(* Logix 5000 project; controller pracainz_ne 1769-L16ER-BB1B rev 30.11; software revision 30.00 *)

TASK MainTask (continuous, watchdog 500 ms) : MainProgram

MODULES
   Local : 1769-L16ER-BB1B (PointIO 0, rev 30.11)
      PF525_1 : vendor 1 type 151 code 9 (Ethernet 192.168.1.76, rev 4.1, Output RPI 20 ms)
          : vendor 1 type 151 code 1566 (DSI 2, rev 1.1)
      pointio : 1734-AENTR (Ethernet 192.168.1.74, rev 5.1, Output RPI 20 ms)
         RTD : 1734-IR2 (PointIO 5, rev 3.1, Input RPI 80 ms)
         input_2 : 1734-IB8 (PointIO 4, rev 3.1)
         input_1 : 1734-IB8 (PointIO 3, rev 3.1)
         potenc : 1734-IE2V (PointIO 6, rev 3.1, Input RPI 80 ms)
         output_2 : 1734-OB8 (PointIO 2, rev 3.1)
         output_1 : 1734-OB8 (PointIO 1, rev 3.1)
      Discrete_IO : Embedded (PointIO 1, rev 30.11, Output RPI 200 ms)
END_MODULES

VAR_GLOBAL   (* controller tags *)
   AUTO_1 : BOOL;
   auto_once : BOOL;
   BELT_CONV_2_0_1_L : BOOL;
   BELT_CONV_2_0_1_U : BOOL;
   BELT_CONV_2_0_2_L : BOOL;
   BELT_CONV_2_0_2_U : BOOL;
   BELT_CONV_2_1_1 : BOOL;
   BELT_CONV_2_1_1_L : BOOL;
   BELT_CONV_2_1_1_U : BOOL;
   BELT_CONV_2_1_2 : BOOL;
   BELT_CONV_2_1_2_L : BOOL;
   BELT_CONV_2_1_2_U : BOOL;
   BELT_CONV_4_0_1_L : BOOL;
   BELT_CONV_4_0_1_U : BOOL;
   BELT_CONV_4_0_2_L : BOOL;
   BELT_CONV_4_0_2_U : BOOL;
   BELT_CONV_4_1_1_L : BOOL;
   BELT_CONV_4_1_1_U : BOOL;
   BELT_CONV_4_1_2_L : BOOL;
   BELT_CONV_4_1_2_U : BOOL;
   BOOL_IN_0 : BOOL;
   BOOL_IN_1 : BOOL;
   BOOL_IN_10 : BOOL;
   BOOL_IN_11 : BOOL := 1;
   BOOL_IN_12 : BOOL := 1;
   BOOL_IN_13 : BOOL := 1;
   BOOL_IN_14 : BOOL := 1;
   BOOL_IN_15 : BOOL := 1;
   BOOL_IN_16 : BOOL;
   BOOL_IN_17 : BOOL;
   BOOL_IN_18 : BOOL := 1;
   BOOL_IN_19 : BOOL := 1;
   BOOL_IN_2 : BOOL;
   BOOL_IN_20 : BOOL;
   BOOL_IN_21 : BOOL;
   BOOL_IN_22 : BOOL := 1;
   BOOL_IN_23 : BOOL;
   BOOL_IN_24 : BOOL;
   BOOL_IN_25 : BOOL;
   BOOL_IN_26 : BOOL := 1;
   BOOL_IN_27 : BOOL := 1;
   BOOL_IN_28 : BOOL;
   BOOL_IN_29 : BOOL := 1;
   BOOL_IN_3 : BOOL;
   BOOL_IN_30 : BOOL := 1;
   BOOL_IN_31 : BOOL := 1;
   BOOL_IN_32 : BOOL := 1;
   BOOL_IN_33 : BOOL := 1;
   BOOL_IN_34 : BOOL;
   BOOL_IN_35 : BOOL;
   BOOL_IN_36 : BOOL;
   BOOL_IN_37 : BOOL;
   BOOL_IN_38 : BOOL := 1;
   BOOL_IN_39 : BOOL := 1;
   BOOL_IN_4 : BOOL;
   BOOL_IN_40 : BOOL := 1;
   BOOL_IN_41 : BOOL;
   BOOL_IN_42 : BOOL;
   BOOL_IN_43 : BOOL;
   BOOL_IN_5 : BOOL;
   BOOL_IN_6 : BOOL;
   BOOL_IN_7 : BOOL;
   BOOL_IN_8 : BOOL := 1;
   BOOL_IN_9 : BOOL;
   BOOL_OUT_0 : BOOL;
   BOOL_OUT_1 : BOOL;
   BOOL_OUT_10 : BOOL;
   BOOL_OUT_11 : BOOL;
   BOOL_OUT_12 : BOOL;
   BOOL_OUT_13 : BOOL;
   BOOL_OUT_14 : BOOL;
   BOOL_OUT_15 : BOOL;
   BOOL_OUT_16 : BOOL;
   BOOL_OUT_17 : BOOL;
   BOOL_OUT_18 : BOOL;
   BOOL_OUT_19 : BOOL;
   BOOL_OUT_2 : BOOL;
   BOOL_OUT_20 : BOOL;
   BOOL_OUT_21 : BOOL;
   BOOL_OUT_22 : BOOL;
   BOOL_OUT_23 : BOOL;
   BOOL_OUT_24 : BOOL;
   BOOL_OUT_25 : BOOL;
   BOOL_OUT_26 : BOOL;
   BOOL_OUT_27 : BOOL;
   BOOL_OUT_28 : BOOL;
   BOOL_OUT_29 : BOOL;
   BOOL_OUT_3 : BOOL;
   BOOL_OUT_30 : BOOL;
   BOOL_OUT_31 : BOOL;
   BOOL_OUT_32 : BOOL;
   BOOL_OUT_33 : BOOL;
   BOOL_OUT_34 : BOOL;
   BOOL_OUT_35 : BOOL := 1;
   BOOL_OUT_36 : BOOL := 1;
   BOOL_OUT_37 : BOOL;
   BOOL_OUT_38 : BOOL;
   BOOL_OUT_39 : BOOL;
   BOOL_OUT_4 : BOOL;
   BOOL_OUT_40 : BOOL;
   BOOL_OUT_41 : BOOL;
   BOOL_OUT_42 : BOOL;
   BOOL_OUT_43 : BOOL;
   BOOL_OUT_44 : BOOL;
   BOOL_OUT_45 : BOOL;
   BOOL_OUT_46 : BOOL;
   BOOL_OUT_47 : BOOL;
   BOOL_OUT_48 : BOOL;
   BOOL_OUT_49 : BOOL := 1;
   BOOL_OUT_5 : BOOL;
   BOOL_OUT_50 : BOOL;
   BOOL_OUT_51 : BOOL;
   BOOL_OUT_52 : BOOL;
   BOOL_OUT_53 : BOOL;
   BOOL_OUT_54 : BOOL;
   BOOL_OUT_55 : BOOL;
   BOOL_OUT_56 : BOOL;
   BOOL_OUT_57 : BOOL;
   BOOL_OUT_58 : BOOL;
   BOOL_OUT_6 : BOOL;
   BOOL_OUT_7 : BOOL;
   BOOL_OUT_8 : BOOL;
   BOOL_OUT_9 : BOOL;
   CHAIN_1 : BOOL;
   CHAIN_1_B : BOOL;
   CHAIN_1_F : BOOL;
   CHAIN_1_L : BOOL;
   CHAIN_1_R : BOOL;
   CHAIN_2 : BOOL;
   CHAIN_2_B : BOOL;
   CHAIN_2_F : BOOL;
   CHAIN_2_L : BOOL;
   CHAIN_2_R : BOOL;
   CLAMPED : BOOL;
   CLAMPED_R : BOOL;
   COUNT_R : DINT;
   dokonczyc : BOOL;
   EMERGENCY_ALL : BOOL := 1;
   END : BOOL;
   END_OF_DAY : BOOL;
   FLOAT_IN_0 : REAL := 1.0;
   FLOAT_IN_1 : REAL := 3.50007;
   FLOAT_IN_2 : REAL := 6.000015;
   FLOAT_IN_3 : REAL := 5.000424;
   FLOAT_IN_4 : REAL := 3.999957;
   FLOAT_IN_5 : REAL := 4.999908;
   FLOAT_IN_6 : REAL;
   FLOAT_OUT_0 : REAL := 6.000015;
   FLOAT_OUT_1 : REAL := 4.999908;
   FLOAT_OUT_2 : REAL := 3.50007;
   FLOAT_OUT_3 : REAL := 3.999957;
   FLOAT_OUT_4 : REAL := 5.000424;
   FLOAT_OUT_5 : REAL;
   FLOAT_OUT_6 : REAL;
   FLOAT_OUT_7 : REAL;
   full_palet : BOOL;
   FULL_PALET_R : BOOL;
   GGG : BOOL;
   height : BOOL;
   height1 : BOOL;
   HHH : BOOL;
   Input_1 : BOOL;
   Input_1_R : BOOL;
   Input_2 : BOOL;
   Input_2_R : BOOL;
   Input_3 : BOOL;
   Input_3_R : BOOL;
   Input_4 : BOOL;
   Input_4_R : BOOL;
   Input_5 : BOOL;
   Input_5_R : BOOL;
   Input_6 : BOOL;
   Input_6_R : BOOL;
   Input_7 : BOOL;
   Input_7_R : BOOL;
   INT_IN_0 : INT;
   INT_IN_1 : INT := 99;
   INT_IN_2 : INT;
   INT_IN_3 : INT;
   INT_OUT_0 : INT;
   koniec : BOOL;
   LATCH_MANUAL : BOOL;
   LEFT_PACK : BOOL;
   LEFT_PACKED : BOOL;
   LEFT_PICK : BOOL;
   LEWA_LINIA : BOOL;
   LEWA_STRONA : BOOL;
   M_01 : BOOL := 1;
   M_02 : BOOL := 1;
   M_03 : BOOL;
   M_04 : BOOL;
   M_05 : BOOL;
   M_06 : BOOL;
   M_07 : BOOL;
   M_08 : BOOL;
   M_09 : BOOL;
   M_10 : BOOL;
   M_11 : BOOL;
   M_12 : BOOL;
   M_13 : BOOL;
   M_14 : BOOL;
   M_15 : BOOL;
   M_16 : BOOL;
   M_17 : BOOL;
   M_18 : BOOL;
   M_19 : BOOL;
   M_20 : BOOL;
   M_21 : INT;
   M_22 : INT;
   M_23 : BOOL;
   M_24 : BOOL;
   M_25 : BOOL := 1;
   M_26 : BOOL;
   M_27 : BOOL;
   M_28 : BOOL;
   M_29 : BOOL;
   M_30 : BOOL;
   M_31 : BOOL;
   M_32 : BOOL;
   M_33 : BOOL;
   M_34 : BOOL;
   M_35 : BOOL;
   M_36 : BOOL;
   M_37 : BOOL;
   M_38 : BOOL;
   M_39 : BOOL;
   M_40 : BOOL;
   M_41 : BOOL;
   M_42 : BOOL;
   M_43 : BOOL;
   M_44 : BOOL;
   M_45 : BOOL;
   M_46 : BOOL;
   M_47 : BOOL;
   MANUAL_ALL : BOOL;
   manual_once : BOOL;
   OSF_03_O : BOOL;
   OSF_03_S : BOOL;
   OSF_05 : BOOL;
   OSF_10_O : BOOL;
   OSF_10_S : BOOL;
   OSF_11_O : BOOL;
   OSF_11_S : BOOL;
   OSFI_01 : DINT;
   OSR_10_O : BOOL;
   OSR_10_S : BOOL := 1;
   OSR_13_O : BOOL;
   OSR_13_S : BOOL;
   OSR_14_O : BOOL;
   OSR_14_S : BOOL := 1;
   OSR_15_O : BOOL;
   OSR_15_S : BOOL;
   OSR_16_O : BOOL;
   OSR_16_S : BOOL;
   OSR_17_O : BOOL;
   OSR_17_S : BOOL;
   OSR_18_O : BOOL;
   OSR_18_S : BOOL := 1;
   OSR_19_O : BOOL;
   OSR_19_S : BOOL;
   OSR_20_O : BOOL;
   OSR_20_S : BOOL;
   OSR_21_O : BOOL;
   OSR_21_S : BOOL := 1;
   OSR_Auto_O : BOOL;
   OSR_Auto_S : BOOL;
   P_P_0_X_D : REAL;
   P_P_0_Y_D : REAL;
   P_P_0_Z_D : REAL;
   PICK : BOOL := 1;
   PRAWA_LINIA : BOOL;
   PRAWA_STRONA : BOOL;
   PUSHER_2 : BOOL;
   READY_L : BOOL;
   READY_R : BOOL;
   Reset : BOOL;
   RESET_1 : BOOL;
   reset_timer : BOOL;
   reset_timer_l : BOOL;
   RIGHT_PACK : BOOL;
   RIGHT_PICK : BOOL;
   ROLL_1 : BOOL;
   ROLL_2 : BOOL;
   ROLL_3 : BOOL;
   ROLL_4 : BOOL;
   ROLL_5 : BOOL;
   ROLL_6 : BOOL;
   ROLL_7 : BOOL;
   START : BOOL;
   START_ALL : BOOL;
   STOP_LEFT : BOOL;
   STOP_RIGHT : BOOL;
   stop_work_timer : TIMER := (PRE := 60000, ACC := 3399, EN := 1, TT := 1);
   stop_work_timer_2 : TIMER := (PRE := 60000);
   stopped_left : BOOL;
   stopped_right : BOOL;
   TASMA_1_P : BOOL;
   TASMA_2_P : BOOL;
   TASMA_5_P : BOOL;
   TASMA_9_P : BOOL;
   TEST_HH : BOOL := 1;
   TIMER_1 : TIMER := (PRE := 800);
   TIMER_2 : TIMER := (PRE := 10000, ACC := 10000, DN := 1);
   TIMER_3_R : TIMER := (PRE := 10000, ACC := 10000, DN := 1);
   TIMER_left : TIMER := (PRE := 100);
   TIMER_LEFT_P_P : TIMER := (PRE := 4000);
   TIMER_PALET : TIMER := (PRE := 500);
   timer_right : TIMER := (PRE := 2000);
   TIMER_RIGHT_P_P : TIMER := (PRE := 4000);
   timer_state_1 : BOOL;
   timer_state_2 : BOOL;
   timer_state_3 : BOOL;
   timer_state_4 : BOOL;
   timer_state_5 : BOOL;
   ton1 : TIMER := (PRE := 2000, ACC := 2000, DN := 1);
   TON1_R : TIMER := (PRE := 2000, ACC := 2000, DN := 1);
   ton2 : TIMER := (PRE := 2000, ACC := 2000, DN := 1);
   TON2_R : TIMER := (PRE := 2000, ACC := 2000, DN := 1);
   ton3 : TIMER := (PRE := 2000);
   ton3_R : TIMER := (PRE := 2000);
   ton4 : TIMER := (PRE := 1000);
   TON4_R : TIMER := (PRE := 1000);
   ton5 : TIMER := (PRE := 3000);
   TON5_R : TIMER := (PRE := 3000);
   ton6 : TIMER := (PRE := 1000);
   TON6_R : TIMER := (PRE := 2000);
   TON7 : TIMER := (PRE := 2000);
   TON7_R : TIMER := (PRE := 2000);
   TONR_01 : FBD_TIMER;
   TONR_02 : FBD_TIMER;
   TONR_03 : FBD_TIMER;
   TONR_04 : FBD_TIMER;
   TONR_05 : FBD_TIMER;
   wait_left : BOOL;
   X0 : REAL := 3.5;
   X1 : REAL := 5.29;
   Y0 : REAL := 6.0;
   Y1 : REAL := 3.8;
   ZNIENNA : BOOL;
END_VAR

PROGRAM MainProgram   (* main routine MainRoutine *)
VAR
   AUTO : ALIAS FOR M_03;
   BELT_CONV_2_0 : ALIAS FOR BOOL_OUT_0;
   BELT_CONV_2_1 : ALIAS FOR BOOL_OUT_1;
   BELT_CONV_2_2 : ALIAS FOR BOOL_OUT_2;
   BELT_CONV_2_3 : ALIAS FOR BOOL_OUT_3;
   BELT_CONV_2_4 : ALIAS FOR BOOL_OUT_4;
   BELT_CONV_2_5 : ALIAS FOR BOOL_OUT_5;
   BELT_CONV_2_6 : ALIAS FOR BOOL_OUT_6;
   BELT_CONV_2_7 : ALIAS FOR BOOL_OUT_7;
   BELT_CONV_2_CCW : ALIAS FOR BOOL_OUT_27;
   BELT_CONV_4_0 : ALIAS FOR BOOL_OUT_8;
   BELT_CONV_4_1 : ALIAS FOR BOOL_OUT_9;
   BELT_CONV_4_2 : ALIAS FOR BOOL_OUT_10;
   BELT_CONV_4_3 : ALIAS FOR BOOL_OUT_11;
   BELT_CONV_CCW_0 : ALIAS FOR BOOL_OUT_23;
   BELT_CONV_CCW_3 : ALIAS FOR BOOL_OUT_24;
   BELT_CONV_CCW_4 : ALIAS FOR BOOL_OUT_25;
   BELT_CONV_CW_0 : ALIAS FOR BOOL_OUT_26;
   BELT_CONV_CW_1 : ALIAS FOR BOOL_OUT_20;
   BELT_CONV_CW_2 : ALIAS FOR BOOL_OUT_21;
   BELT_CONV_CW_5 : ALIAS FOR BOOL_OUT_22;
   BTN_RESET : ALIAS FOR BOOL_IN_34;
   BTN_START : ALIAS FOR BOOL_IN_35;
   BTN_STOP : ALIAS FOR BOOL_IN_38;
   CAP_SEN_0 : ALIAS FOR BOOL_IN_0;
   CAP_SEN_1 : ALIAS FOR BOOL_IN_1;
   CAP_SEN_2 : ALIAS FOR BOOL_IN_2;
   CAP_SEN_3 : ALIAS FOR BOOL_IN_3;
   CHAIN_0_LEFT : ALIAS FOR BOOL_OUT_16;
   CHAIN_0_N : ALIAS FOR BOOL_OUT_13;
   CHAIN_0_P : ALIAS FOR BOOL_OUT_12;
   CHAIN_0_RIGHT : ALIAS FOR BOOL_OUT_18;
   CHAIN_1_LEFT : ALIAS FOR BOOL_OUT_17;
   CHAIN_1_N : ALIAS FOR BOOL_OUT_15;
   CHAIN_1_P : ALIAS FOR BOOL_OUT_14;
   CHAIN_1_RIGHT : ALIAS FOR BOOL_OUT_19;
   CNC_0_START : ALIAS FOR BOOL_OUT_38;
   CNC_1_START : ALIAS FOR BOOL_OUT_40;
   CNC_RESET : BOOL;
   CNC_START_1 : BOOL;
   CNC_STOP_1 : BOOL;
   COUNT : DINT;
   DIFF_SEN_0 : ALIAS FOR BOOL_IN_4;
   DIFF_SEN_1 : ALIAS FOR BOOL_IN_5;
   DIFF_SEN_2 : ALIAS FOR BOOL_IN_6;
   DIFF_SEN_3 : ALIAS FOR BOOL_IN_7;
   DIFF_SEN_4 : ALIAS FOR BOOL_IN_8;
   EMERGENCY : ALIAS FOR BOOL_IN_33;
   emergency_disp : BOOL;
   EMIT_0 : ALIAS FOR BOOL_OUT_28;
   EMIT_1 : ALIAS FOR BOOL_OUT_29;
   EMIT_2 : ALIAS FOR BOOL_OUT_30;
   EMIT_3 : ALIAS FOR BOOL_OUT_31;
   FREQUENCY : INT := 3000;
   GREEN_B : ALIAS FOR M_22;
   GREEN_L : ALIAS FOR M_21;
   koniecpracy : ALIAS FOR koniec;
   MACH_CEN_0_LIDS : ALIAS FOR BOOL_OUT_41;
   MACH_CEN_0_PROGRESS : ALIAS FOR INT_IN_0;
   MACH_CEN_0_RESET : ALIAS FOR BOOL_OUT_39;
   MACH_CEN_0_START : ALIAS FOR BOOL_OUT_37;
   MACH_CEN_0_STOP : ALIAS FOR BOOL_OUT_35;
   MACH_CEN_1_LIDS : ALIAS FOR BOOL_OUT_42;
   MACH_CEN_1_PROGRESS : ALIAS FOR INT_IN_1;
   MACH_CEN_1_RESET : ALIAS FOR BOOL_OUT_40;
   MACH_CEN_1_START : ALIAS FOR BOOL_OUT_38;
   MACH_CEN_1_STOP : ALIAS FOR BOOL_OUT_36;
   MACHI_CE_0_BUSY : ALIAS FOR BOOL_IN_14;
   MACHI_CE_0_ERR : ALIAS FOR BOOL_IN_16;
   MACHI_CE_0_OPEN : ALIAS FOR BOOL_IN_12;
   MACHI_CE_1_BUSY : ALIAS FOR BOOL_IN_15;
   MACHI_CE_1_ERR : ALIAS FOR BOOL_IN_17;
   MACHI_CE_1_OPEN : ALIAS FOR BOOL_IN_13;
   MACHINE_X : REAL;
   MACHINE_Y : REAL;
   MACHINE_Z : REAL;
   MANUAL : ALIAS FOR M_04;
   manual_disp : BOOL := 1;
   MOVE : ALIAS FOR M_16;
   NOT_BLUE : ALIAS FOR M_24;
   NOT_GREEN : ALIAS FOR M_23;
   OSF_01_O : ALIAS FOR M_07;
   OSF_01_S : ALIAS FOR M_06;
   OSF_02_O : ALIAS FOR M_11;
   OSF_02_S : ALIAS FOR M_10;
   OSF_03_O : ALIAS FOR M_05;
   OSF_03_S : ALIAS FOR M_25;
   OSF_04_O : ALIAS FOR M_26;
   OSF_04_S : ALIAS FOR M_27;
   OSF_05_O : ALIAS FOR M_28;
   OSF_05_S : ALIAS FOR M_29;
   OSF_06_O : ALIAS FOR M_30;
   OSF_06_S : ALIAS FOR M_31;
   OSF_07_O : ALIAS FOR M_32;
   OSF_07_S : ALIAS FOR M_30;
   OSF_08_O : ALIAS FOR M_41;
   OSF_08_S : ALIAS FOR M_42;
   OSF_09_O : BOOL;
   OSF_09_S : BOOL := 1;
   OSR_01_O : ALIAS FOR M_09;
   OSR_01_S : ALIAS FOR M_08;
   OSR_02_O : ALIAS FOR M_13;
   OSR_02_S : ALIAS FOR M_12;
   OSR_03_O : ALIAS FOR M_17;
   OSR_03_S : ALIAS FOR M_18;
   OSR_04_O : ALIAS FOR M_19;
   OSR_04_S : ALIAS FOR M_20;
   OSR_05_O : ALIAS FOR M_14;
   OSR_05_S : ALIAS FOR M_15;
   OSR_06_O : ALIAS FOR M_33;
   OSR_06_S : ALIAS FOR M_34;
   OSR_07_O : ALIAS FOR M_35;
   OSR_07_S : ALIAS FOR M_36;
   OSR_08_O : ALIAS FOR M_37;
   OSR_08_S : ALIAS FOR M_38;
   OSR_09_O : ALIAS FOR M_39;
   OSR_09_S : ALIAS FOR M_40;
   P_P_0_C_LIMIT : ALIAS FOR BOOL_IN_18;
   P_P_0_CP : ALIAS FOR BOOL_OUT_43;
   P_P_0_DETE : ALIAS FOR BOOL_IN_20;
   P_P_0_GRAB : ALIAS FOR BOOL_OUT_45;
   P_P_0_X : ALIAS FOR FLOAT_OUT_2;
   P_P_0_X_POSITION : ALIAS FOR FLOAT_IN_1;
   P_P_0_Y : ALIAS FOR FLOAT_OUT_0;
   P_P_0_Y_POSITION : ALIAS FOR FLOAT_IN_2;
   P_P_0_Z : ALIAS FOR FLOAT_OUT_4;
   P_P_0_Z_POSITION : ALIAS FOR FLOAT_IN_3;
   P_P_1_C_LIMIT : ALIAS FOR BOOL_IN_19;
   P_P_1_CP : ALIAS FOR BOOL_OUT_44;
   P_P_1_DETE : ALIAS FOR BOOL_IN_21;
   P_P_1_GRAB : ALIAS FOR BOOL_OUT_46;
   P_P_1_X : ALIAS FOR FLOAT_OUT_3;
   P_P_1_X_D : REAL := 4.0;
   P_P_1_X_POSITION : ALIAS FOR FLOAT_IN_4;
   P_P_1_Y : ALIAS FOR FLOAT_OUT_1;
   P_P_1_Y_D : REAL := 5.0;
   P_P_1_Y_POSITION : ALIAS FOR FLOAT_IN_5;
   P_P_1_Z : ALIAS FOR FLOAT_OUT_5;
   P_P_1_Z_D : REAL := 5.0;
   P_P_1_Z_POSITION : ALIAS FOR FLOAT_IN_6;
   PUSH_0 : ALIAS FOR BOOL_OUT_47;
   PUSH_0_BACK : ALIAS FOR BOOL_IN_22;
   PUSH_0_FRONT : ALIAS FOR BOOL_IN_23;
   PUSH_1 : ALIAS FOR BOOL_OUT_48;
   PUSH_1_BACK : ALIAS FOR BOOL_IN_39;
   PUSH_1_FRONT : ALIAS FOR BOOL_IN_24;
   PUSHER_1 : BOOL;
   REMOVER : ALIAS FOR BOOL_OUT_49;
   RETRO_SEN_0 : ALIAS FOR BOOL_IN_25;
   RETRO_SEN_1 : ALIAS FOR BOOL_IN_26;
   RETRO_SEN_2 : ALIAS FOR BOOL_IN_27;
   RETRO_SEN_3 : ALIAS FOR BOOL_IN_28;
   RETRO_SEN_4 : ALIAS FOR BOOL_IN_29;
   RETRO_SEN_5 : ALIAS FOR BOOL_IN_30;
   RETRO_SEN_6 : ALIAS FOR BOOL_IN_31;
   RETRO_SEN_7 : ALIAS FOR BOOL_IN_32;
   ROLL_4_0 : ALIAS FOR BOOL_OUT_50;
   ROLL_4_1 : ALIAS FOR BOOL_OUT_51;
   ROLL_4_2 : ALIAS FOR BOOL_OUT_52;
   ROLL_6_0 : ALIAS FOR BOOL_OUT_53;
   ROLL_6_1 : ALIAS FOR BOOL_OUT_54;
   start_disp : BOOL := 1;
   STOP_ALL : ALIAS FOR M_02;
   stop_disp : BOOL;
   STOP_EMIT : ALIAS FOR M_01;
   TASMA_1 : BOOL;
   TASMA_10 : BOOL;
   TASMA_2 : BOOL;
   TASMA_3 : BOOL;
   TASMA_4 : BOOL;
   TASMA_5 : BOOL;
   TASMA_6 : BOOL;
   TASMA_7 : BOOL;
   TASMA_8 : BOOL;
   TASMA_9 : BOOL;
   VISION_SEN_0 : ALIAS FOR INT_IN_2;
   VISION_SEN_1 : ALIAS FOR INT_IN_3;
END_VAR

ROUTINE MainRoutine   (* ladder *)
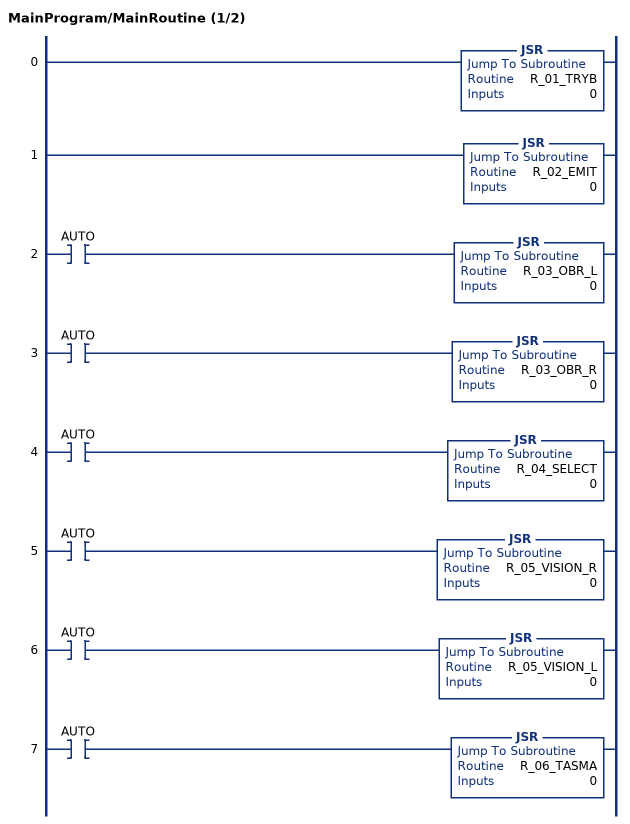
   0: JSR(R_01_TRYB,0);
   1: JSR(R_02_EMIT,0);
   2: XIC(AUTO)JSR(R_03_OBR_L,0);
   3: XIC(AUTO)JSR(R_03_OBR_R,0);
   4: XIC(AUTO)JSR(R_04_SELECT,0);
   5: XIC(AUTO)JSR(R_05_VISION_R,0);
   6: XIC(AUTO)JSR(R_05_VISION_L,0);
   7: XIC(AUTO)JSR(R_06_TASMA,0);
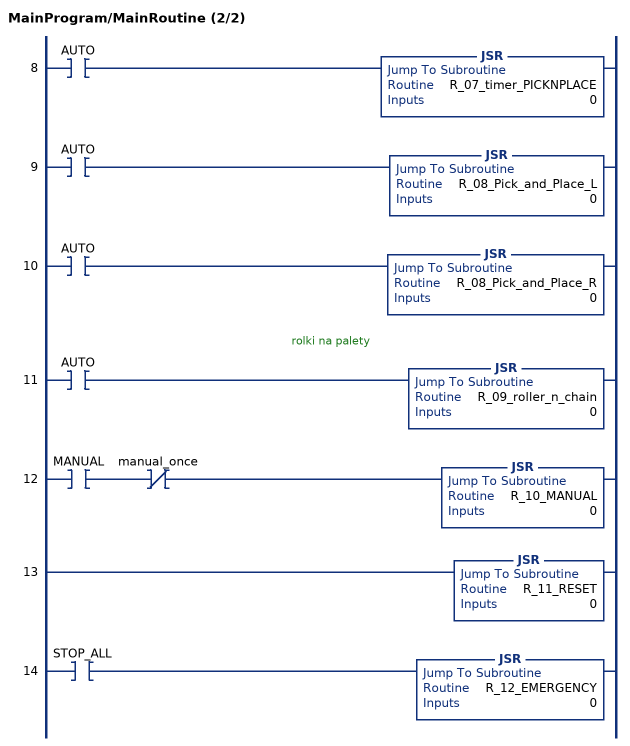
   8: XIC(AUTO)JSR(R_07_timer_PICKNPLACE,0);
   9: XIC(AUTO)JSR(R_08_Pick_and_Place_L,0);
   10: XIC(AUTO)JSR(R_08_Pick_and_Place_R,0);
   // rolki na palety
   11: XIC(AUTO)JSR(R_09_roller_n_chain,0);
   12: XIC(MANUAL)XIO(manual_once)JSR(R_10_MANUAL,0);
   13: JSR(R_11_RESET,0);
   14: XIC(STOP_ALL)JSR(R_12_EMERGENCY,0);
END_ROUTINE

ROUTINE R_01_TRYB   (* ladder *)
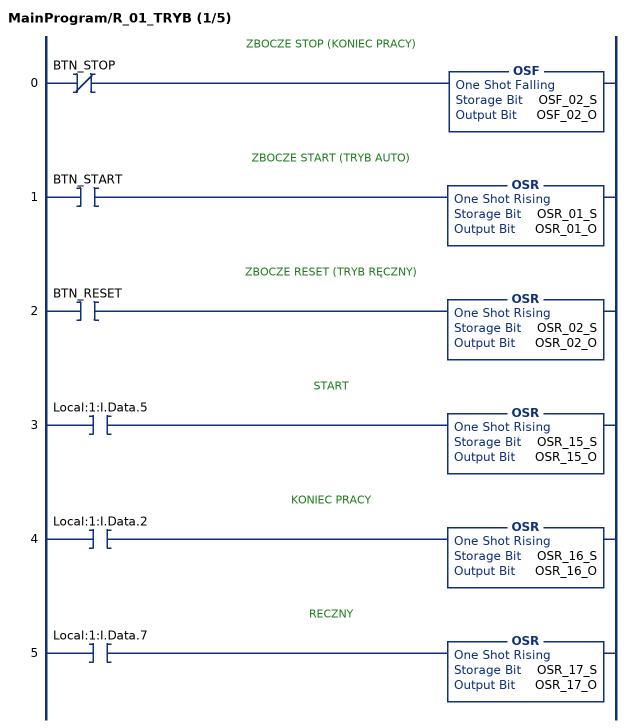
   // ZBOCZE STOP (KONIEC PRACY)
   0: XIO(BTN_STOP)OSF(OSF_02_S,OSF_02_O);
   // ZBOCZE START (TRYB AUTO)
   1: XIC(BTN_START)OSR(OSR_01_S,OSR_01_O);
   // ZBOCZE RESET (TRYB RĘCZNY)
   2: XIC(BTN_RESET)OSR(OSR_02_S,OSR_02_O);
   // START
   3: XIC(Local:1:I.Data.5)OSR(OSR_15_S,OSR_15_O);
   // KONIEC PRACY
   4: XIC(Local:1:I.Data.2)OSR(OSR_16_S,OSR_16_O);
   // RECZNY
   5: XIC(Local:1:I.Data.7)OSR(OSR_17_S,OSR_17_O);
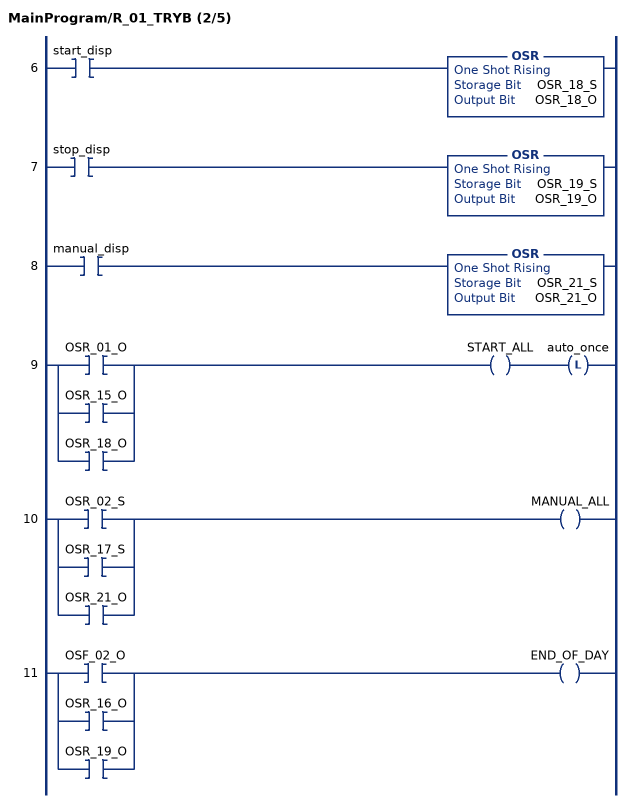
   6: XIC(start_disp)OSR(OSR_18_S,OSR_18_O);
   7: XIC(stop_disp)OSR(OSR_19_S,OSR_19_O);
   8: XIC(manual_disp)OSR(OSR_21_S,OSR_21_O);
   9: [XIC(OSR_01_O) ,XIC(OSR_15_O) ,XIC(OSR_18_O) ]OTE(START_ALL)OTL(auto_once);
   10: [XIC(OSR_02_S) ,XIC(OSR_17_S) ,XIC(OSR_21_O) ]OTE(MANUAL_ALL);
   11: [XIC(OSF_02_O) ,XIC(OSR_16_O) ,XIC(OSR_19_O) ]OTE(END_OF_DAY);
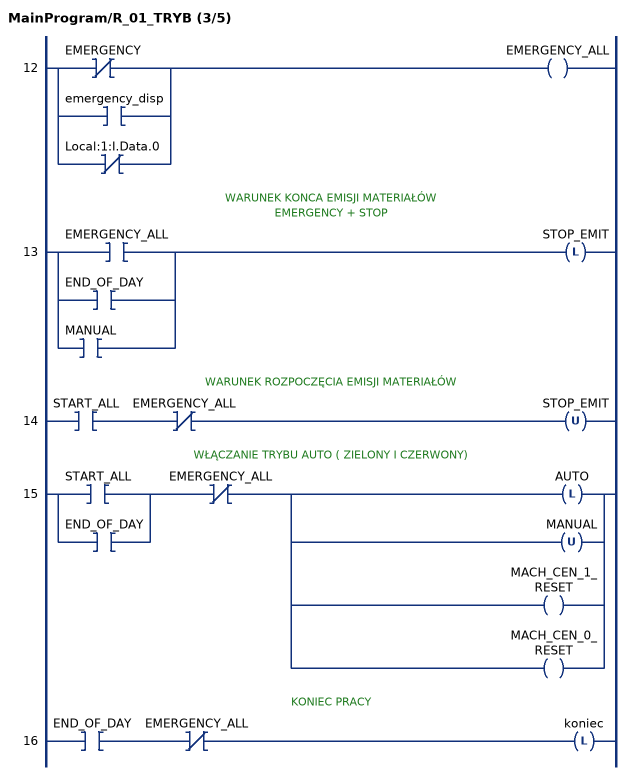
   12: [XIO(EMERGENCY) ,XIC(emergency_disp) ,XIO(Local:1:I.Data.0) ]OTE(EMERGENCY_ALL);
   // WARUNEK KONCA EMISJI MATERIAŁÓW
   // EMERGENCY + STOP
   13: [XIC(EMERGENCY_ALL) ,XIC(END_OF_DAY) ,XIC(MANUAL) ]OTL(STOP_EMIT);
   // WARUNEK ROZPOCZĘCIA EMISJI MATERIAŁÓW
   14: XIC(START_ALL)XIO(EMERGENCY_ALL)OTU(STOP_EMIT);
   // WŁĄCZANIE TRYBU AUTO ( ZIELONY I CZERWONY)
   15: [XIC(START_ALL) ,XIC(END_OF_DAY) ]XIO(EMERGENCY_ALL)[OTL(AUTO) ,OTU(MANUAL) ,OTE(MACH_CEN_1_RESET) ,OTE(MACH_CEN_0_RESET) ];
   // KONIEC PRACY
   16: XIC(END_OF_DAY)XIO(EMERGENCY_ALL)OTL(koniec);
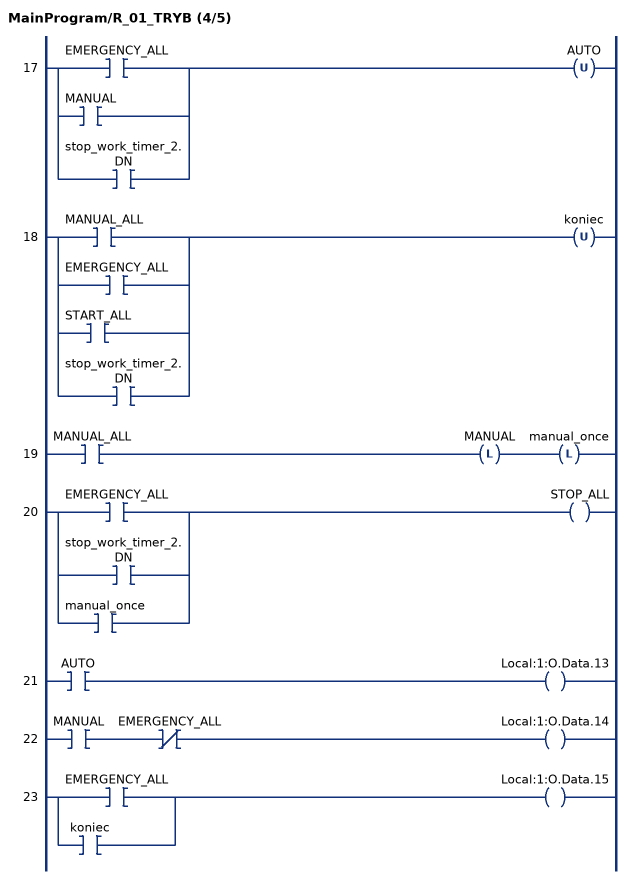
   17: [XIC(EMERGENCY_ALL) ,XIC(MANUAL) ,XIC(stop_work_timer_2.DN) ]OTU(AUTO);
   18: [XIC(MANUAL_ALL) ,XIC(EMERGENCY_ALL) ,XIC(START_ALL) ,XIC(stop_work_timer_2.DN) ]OTU(koniec);
   19: XIC(MANUAL_ALL)OTL(MANUAL)OTL(manual_once);
   20: [XIC(EMERGENCY_ALL) ,XIC(stop_work_timer_2.DN) ,XIC(manual_once) ]OTE(STOP_ALL);
   21: XIC(AUTO)OTE(Local:1:O.Data.13);
   22: XIC(MANUAL)XIO(EMERGENCY_ALL)OTE(Local:1:O.Data.14);
   23: [XIC(EMERGENCY_ALL) ,XIC(koniec) ]OTE(Local:1:O.Data.15);
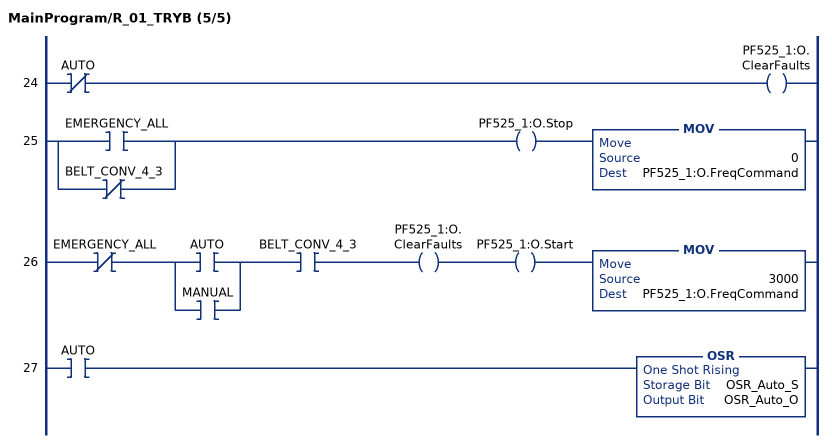
   24: XIO(AUTO)OTE(PF525_1:O.ClearFaults);
   25: [XIC(EMERGENCY_ALL) ,XIO(BELT_CONV_4_3) ]OTE(PF525_1:O.Stop)MOV(0,PF525_1:O.FreqCommand);
   26: XIO(EMERGENCY_ALL)[XIC(AUTO) ,XIC(MANUAL) ]XIC(BELT_CONV_4_3)OTE(PF525_1:O.ClearFaults)OTE(PF525_1:O.Start)MOV(3000,PF525_1:O.FreqCommand);
   27: XIC(AUTO)OSR(OSR_Auto_S,OSR_Auto_O);
END_ROUTINE

ROUTINE R_02_EMIT   (* ladder *)
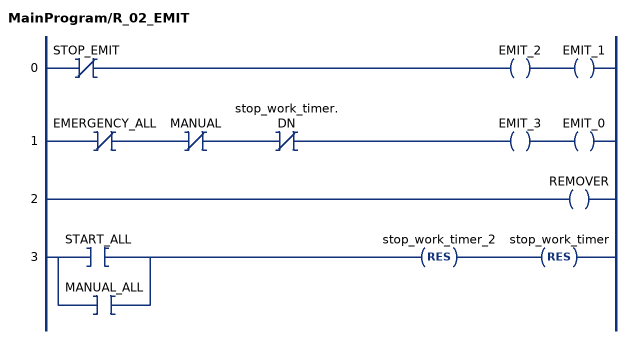
   0: XIO(STOP_EMIT)OTE(EMIT_2)OTE(EMIT_1);
   1: XIO(EMERGENCY_ALL)XIO(MANUAL)XIO(stop_work_timer.DN)OTE(EMIT_3)OTE(EMIT_0);
   2: OTE(REMOVER);
   3: [XIC(START_ALL) ,XIC(MANUAL_ALL) ]RES(stop_work_timer_2)RES(stop_work_timer);
END_ROUTINE

ROUTINE R_03_OBR_L   (* ladder *)
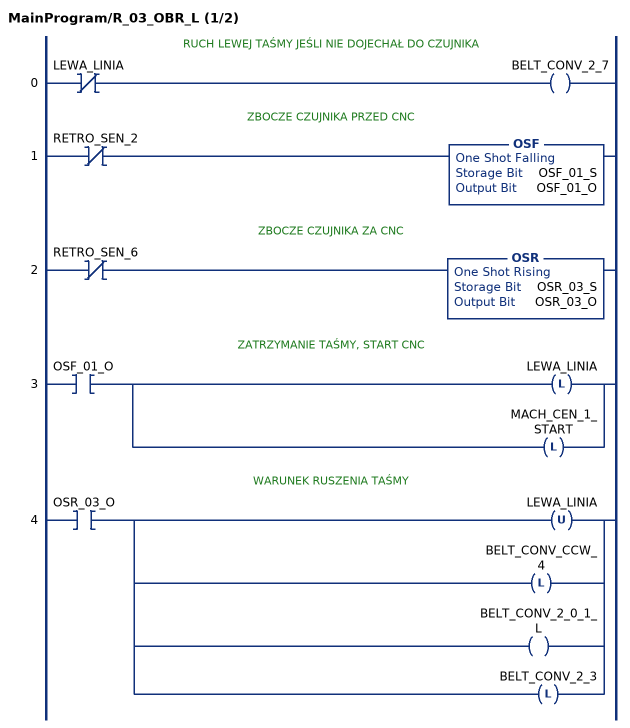
   // RUCH LEWEJ TAŚMY JEŚLI NIE DOJECHAŁ DO CZUJNIKA
   0: XIO(LEWA_LINIA)OTE(BELT_CONV_2_7);
   // ZBOCZE CZUJNIKA PRZED CNC
   1: XIO(RETRO_SEN_2)OSF(OSF_01_S,OSF_01_O);
   // ZBOCZE CZUJNIKA ZA CNC
   2: XIO(RETRO_SEN_6)OSR(OSR_03_S,OSR_03_O);
   // ZATRZYMANIE TAŚMY, START CNC
   3: XIC(OSF_01_O)[OTL(LEWA_LINIA) ,OTL(MACH_CEN_1_START) ];
   // WARUNEK RUSZENIA TAŚMY
   4: XIC(OSR_03_O)[OTU(LEWA_LINIA) ,OTL(BELT_CONV_CCW_4) ,OTE(BELT_CONV_2_0_1_L) ,OTL(BELT_CONV_2_3) ];
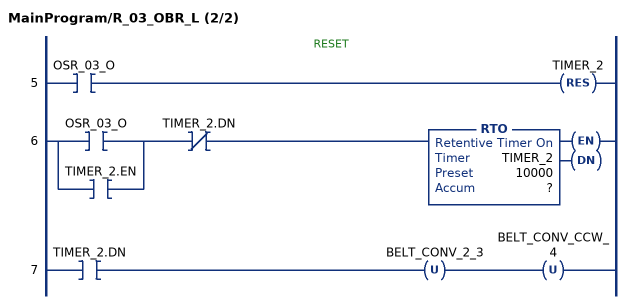
   // RESET
   5: XIC(OSR_03_O)RES(TIMER_2);
   6: [XIC(OSR_03_O) ,XIC(TIMER_2.EN) ]XIO(TIMER_2.DN)RTO(TIMER_2,?,?);
   7: XIC(TIMER_2.DN)OTU(BELT_CONV_2_3)OTU(BELT_CONV_CCW_4);
END_ROUTINE

ROUTINE R_03_OBR_R   (* ladder *)
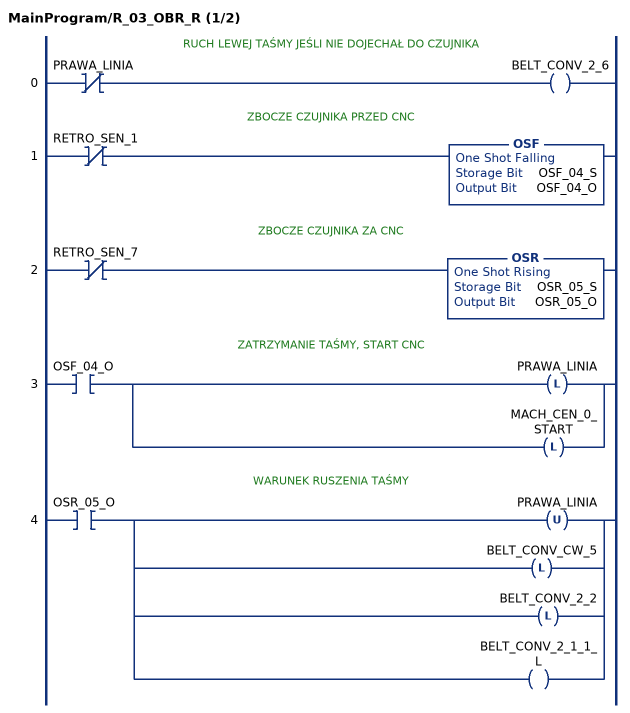
   // RUCH LEWEJ TAŚMY JEŚLI NIE DOJECHAŁ DO CZUJNIKA
   0: XIO(PRAWA_LINIA)OTE(BELT_CONV_2_6);
   // ZBOCZE CZUJNIKA PRZED CNC
   1: XIO(RETRO_SEN_1)OSF(OSF_04_S,OSF_04_O);
   // ZBOCZE CZUJNIKA ZA CNC
   2: XIO(RETRO_SEN_7)OSR(OSR_05_S,OSR_05_O);
   // ZATRZYMANIE TAŚMY, START CNC
   3: XIC(OSF_04_O)[OTL(PRAWA_LINIA) ,OTL(MACH_CEN_0_START) ];
   // WARUNEK RUSZENIA TAŚMY
   4: XIC(OSR_05_O)[OTU(PRAWA_LINIA) ,OTL(BELT_CONV_CW_5) ,OTL(BELT_CONV_2_2) ,OTE(BELT_CONV_2_1_1_L) ];
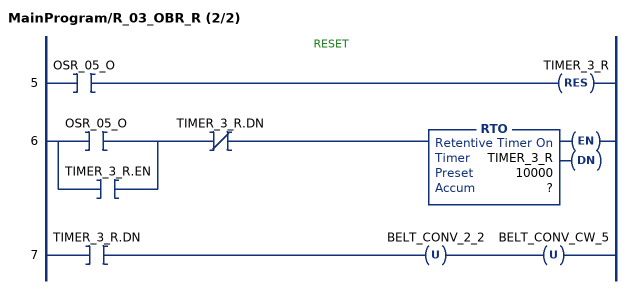
   // RESET
   5: XIC(OSR_05_O)RES(TIMER_3_R);
   6: [XIC(OSR_05_O) ,XIC(TIMER_3_R.EN) ]XIO(TIMER_3_R.DN)RTO(TIMER_3_R,?,?);
   7: XIC(TIMER_3_R.DN)OTU(BELT_CONV_2_2)OTU(BELT_CONV_CW_5);
END_ROUTINE

ROUTINE R_04_SELECT   (* ladder *)
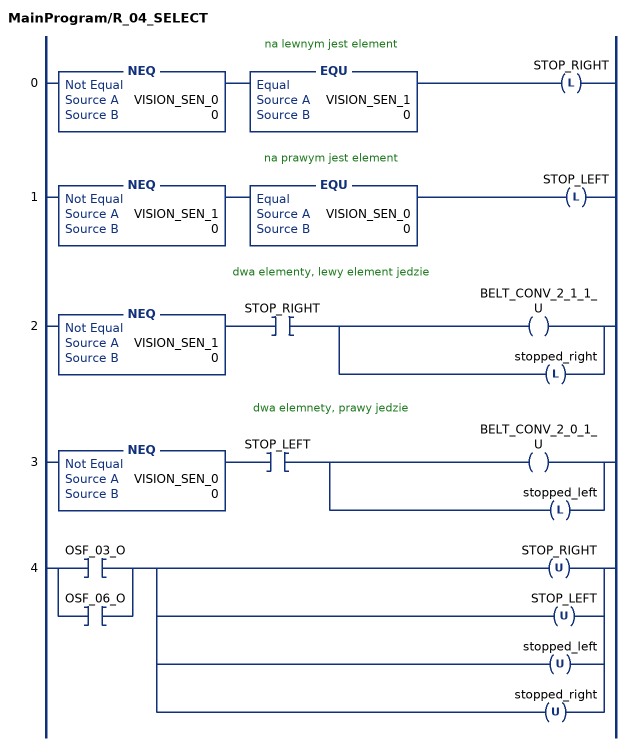
   // na lewnym jest element
   0: NEQ(VISION_SEN_0,0)EQU(VISION_SEN_1,0)OTL(STOP_RIGHT);
   // na prawym jest element
   1: NEQ(VISION_SEN_1,0)EQU(VISION_SEN_0,0)OTL(STOP_LEFT);
   // dwa elementy, lewy element jedzie
   2: NEQ(VISION_SEN_1,0)XIC(STOP_RIGHT)[OTE(BELT_CONV_2_1_1_U) ,OTL(stopped_right) ];
   // dwa elemnety, prawy jedzie
   3: NEQ(VISION_SEN_0,0)XIC(STOP_LEFT)[OTE(BELT_CONV_2_0_1_U) ,OTL(stopped_left) ];
   4: [XIC(OSF_03_O) ,XIC(OSF_06_O) ][OTU(STOP_RIGHT) ,OTU(STOP_LEFT) ,OTU(stopped_left) ,OTU(stopped_right) ];
END_ROUTINE

ROUTINE R_05_VISION_L   (* ladder *)
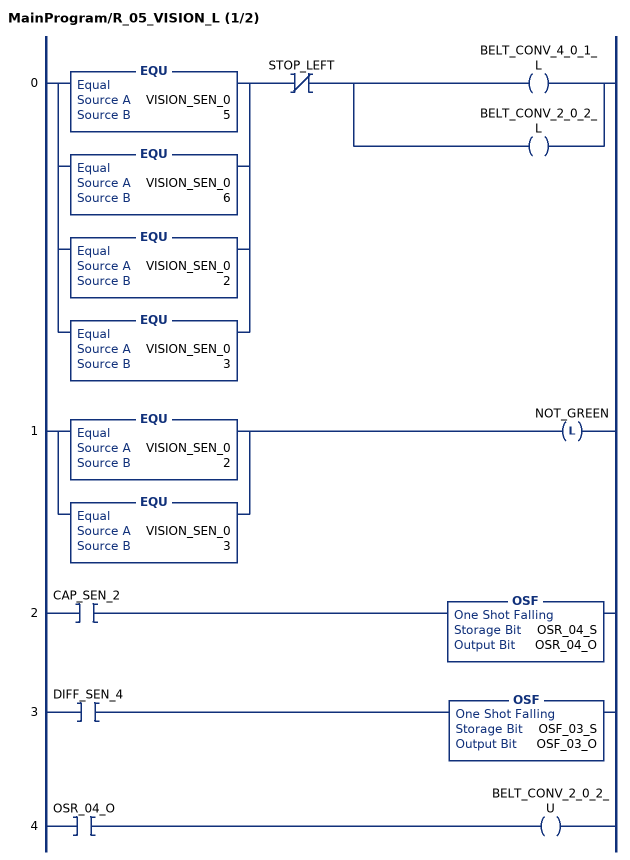
   0: [EQU(VISION_SEN_0,5) ,EQU(VISION_SEN_0,6) ,EQU(VISION_SEN_0,2) ,EQU(VISION_SEN_0,3) ]XIO(STOP_LEFT)[OTE(BELT_CONV_4_0_1_L) ,OTE(BELT_CONV_2_0_2_L) ];
   1: [EQU(VISION_SEN_0,2) ,EQU(VISION_SEN_0,3) ]OTL(NOT_GREEN);
   2: XIC(CAP_SEN_2)OSF(OSR_04_S,OSR_04_O);
   3: XIC(DIFF_SEN_4)OSF(OSF_03_S,OSF_03_O);
   4: XIC(OSR_04_O)OTE(BELT_CONV_2_0_2_U);
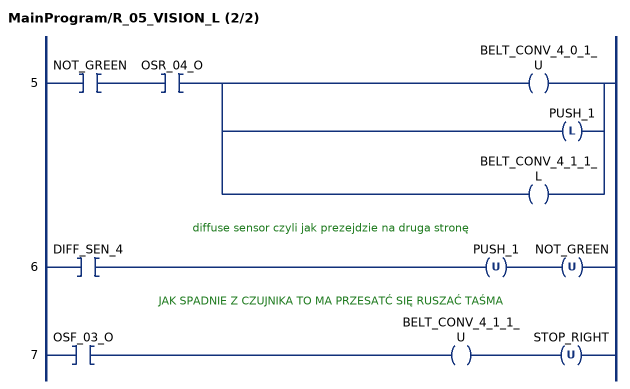
   5: XIC(NOT_GREEN)XIC(OSR_04_O)[OTE(BELT_CONV_4_0_1_U) ,OTL(PUSH_1) ,OTE(BELT_CONV_4_1_1_L) ];
   // diffuse sensor czyli jak prezejdzie na druga stronę
   6: XIC(DIFF_SEN_4)OTU(PUSH_1)OTU(NOT_GREEN);
   // JAK SPADNIE Z CZUJNIKA TO MA PRZESATĆ SIĘ RUSZAĆ TAŚMA
   7: XIC(OSF_03_O)OTE(BELT_CONV_4_1_1_U)OTU(STOP_RIGHT);
END_ROUTINE

ROUTINE R_05_VISION_R   (* ladder *)
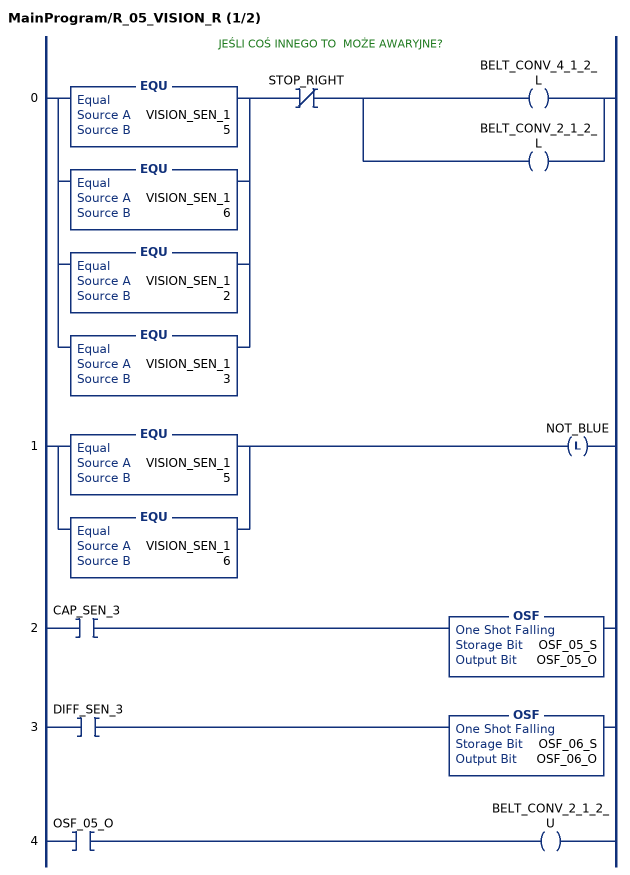
   // JEŚLI COŚ INNEGO TO  MOŻE AWARYJNE?
   0: [EQU(VISION_SEN_1,5) ,EQU(VISION_SEN_1,6) ,EQU(VISION_SEN_1,2) ,EQU(VISION_SEN_1,3) ]XIO(STOP_RIGHT)[OTE(BELT_CONV_4_1_2_L) ,OTE(BELT_CONV_2_1_2_L) ];
   1: [EQU(VISION_SEN_1,5) ,EQU(VISION_SEN_1,6) ]OTL(NOT_BLUE);
   2: XIC(CAP_SEN_3)OSF(OSF_05_S,OSF_05_O);
   3: XIC(DIFF_SEN_3)OSF(OSF_06_S,OSF_06_O);
   4: XIC(OSF_05_O)OTE(BELT_CONV_2_1_2_U);
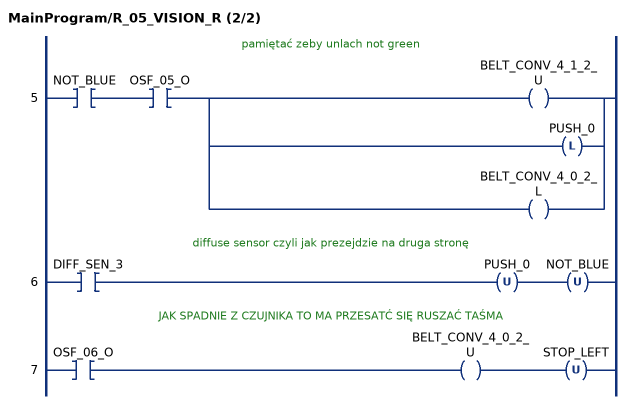
   // pamiętać zeby unlach not green
   5: XIC(NOT_BLUE)XIC(OSF_05_O)[OTE(BELT_CONV_4_1_2_U) ,OTL(PUSH_0) ,OTE(BELT_CONV_4_0_2_L) ];
   // diffuse sensor czyli jak prezejdzie na druga stronę
   6: XIC(DIFF_SEN_3)OTU(PUSH_0)OTU(NOT_BLUE);
   // JAK SPADNIE Z CZUJNIKA TO MA PRZESATĆ SIĘ RUSZAĆ TAŚMA
   7: XIC(OSF_06_O)OTE(BELT_CONV_4_0_2_U)OTU(STOP_LEFT);
END_ROUTINE

ROUTINE R_06_TASMA   (* ladder *)
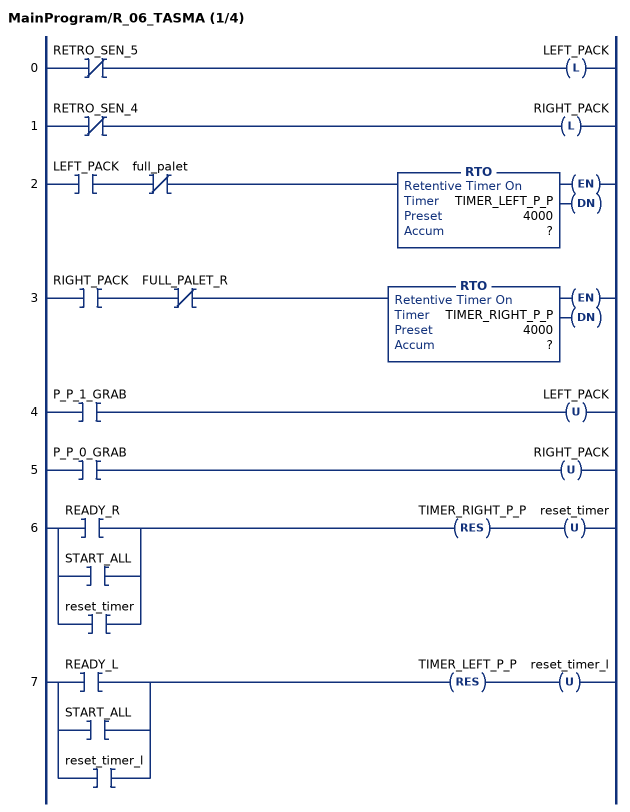
   0: XIO(RETRO_SEN_5)OTL(LEFT_PACK);
   1: XIO(RETRO_SEN_4)OTL(RIGHT_PACK);
   2: XIC(LEFT_PACK)XIO(full_palet)RTO(TIMER_LEFT_P_P,?,?);
   3: XIC(RIGHT_PACK)XIO(FULL_PALET_R)RTO(TIMER_RIGHT_P_P,?,?);
   4: XIC(P_P_1_GRAB)OTU(LEFT_PACK);
   5: XIC(P_P_0_GRAB)OTU(RIGHT_PACK);
   6: [XIC(READY_R) ,XIC(START_ALL) ,XIC(reset_timer) ]RES(TIMER_RIGHT_P_P)OTU(reset_timer);
   7: [XIC(READY_L) ,XIC(START_ALL) ,XIC(reset_timer_l) ]RES(TIMER_LEFT_P_P)OTU(reset_timer_l);
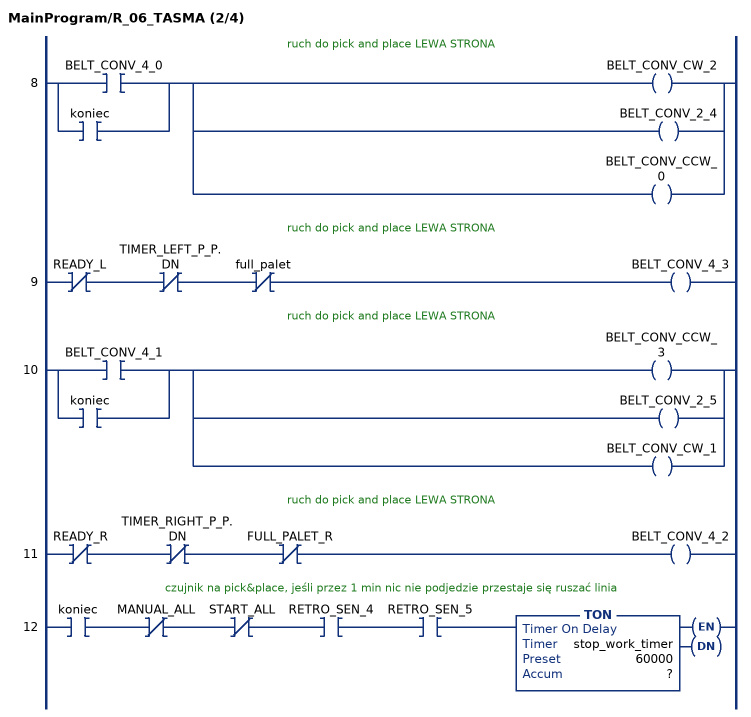
   // ruch do pick and place LEWA STRONA
   8: [XIC(BELT_CONV_4_0) ,XIC(koniec) ][OTE(BELT_CONV_CW_2) ,OTE(BELT_CONV_2_4) ,OTE(BELT_CONV_CCW_0) ];
   // ruch do pick and place LEWA STRONA
   9: XIO(READY_L)XIO(TIMER_LEFT_P_P.DN)XIO(full_palet)OTE(BELT_CONV_4_3);
   // ruch do pick and place LEWA STRONA
   10: [XIC(BELT_CONV_4_1) ,XIC(koniec) ][OTE(BELT_CONV_CCW_3) ,OTE(BELT_CONV_2_5) ,OTE(BELT_CONV_CW_1) ];
   // ruch do pick and place LEWA STRONA
   11: XIO(READY_R)XIO(TIMER_RIGHT_P_P.DN)XIO(FULL_PALET_R)OTE(BELT_CONV_4_2);
   // czujnik na pick&place, jeśli przez 1 min nic nie podjedzie przestaje się ruszać linia
   12: XIC(koniec)XIO(MANUAL_ALL)XIO(START_ALL)XIC(RETRO_SEN_4)XIC(RETRO_SEN_5)TON(stop_work_timer,?,?);
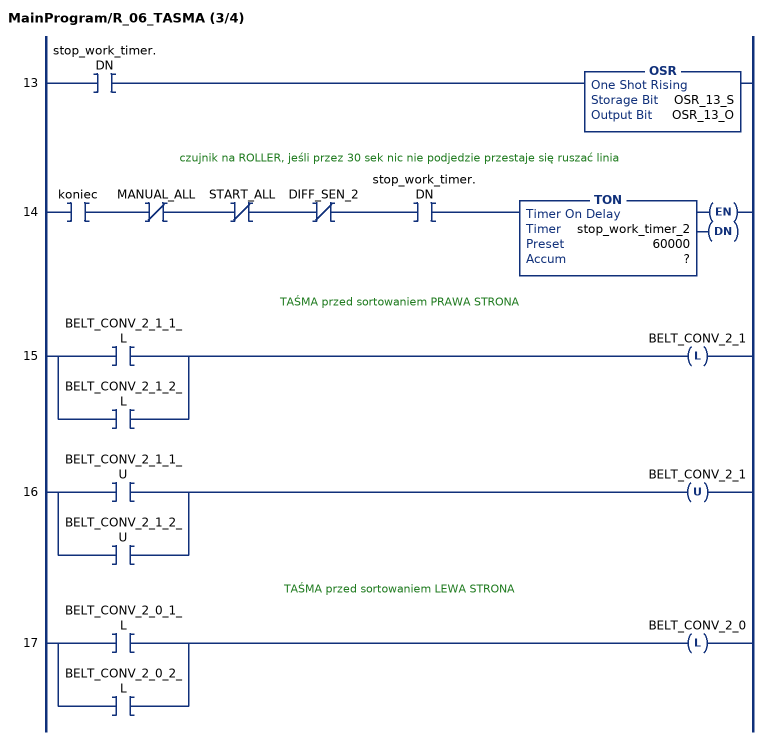
   13: XIC(stop_work_timer.DN)OSR(OSR_13_S,OSR_13_O);
   // czujnik na ROLLER, jeśli przez 30 sek nic nie podjedzie przestaje się ruszać linia
   14: XIC(koniec)XIO(MANUAL_ALL)XIO(START_ALL)XIO(DIFF_SEN_2)XIC(stop_work_timer.DN)TON(stop_work_timer_2,?,?);
   // TAŚMA przed sortowaniem PRAWA STRONA
   15: [XIC(BELT_CONV_2_1_1_L) ,XIC(BELT_CONV_2_1_2_L) ]OTL(BELT_CONV_2_1);
   16: [XIC(BELT_CONV_2_1_1_U) ,XIC(BELT_CONV_2_1_2_U) ]OTU(BELT_CONV_2_1);
   // TAŚMA przed sortowaniem LEWA STRONA
   17: [XIC(BELT_CONV_2_0_1_L) ,XIC(BELT_CONV_2_0_2_L) ]OTL(BELT_CONV_2_0);
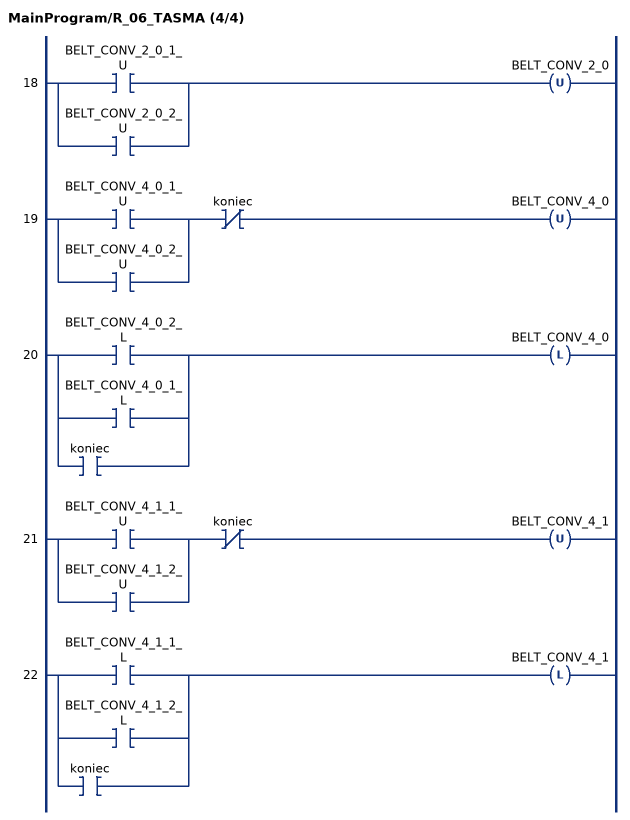
   18: [XIC(BELT_CONV_2_0_1_U) ,XIC(BELT_CONV_2_0_2_U) ]OTU(BELT_CONV_2_0);
   19: [XIC(BELT_CONV_4_0_1_U) ,XIC(BELT_CONV_4_0_2_U) ]XIO(koniec)OTU(BELT_CONV_4_0);
   20: [XIC(BELT_CONV_4_0_2_L) ,XIC(BELT_CONV_4_0_1_L) ,XIC(koniec) ]OTL(BELT_CONV_4_0);
   21: [XIC(BELT_CONV_4_1_1_U) ,XIC(BELT_CONV_4_1_2_U) ]XIO(koniec)OTU(BELT_CONV_4_1);
   22: [XIC(BELT_CONV_4_1_1_L) ,XIC(BELT_CONV_4_1_2_L) ,XIC(koniec) ]OTL(BELT_CONV_4_1);
END_ROUTINE
